// TIA Portal V20 export
TYPE "UDT_Service_ValueDefinition"
   STRUCT
      indexMTP : Int;   // Index of value / MTP Index of value
      indexIO : Int;   // Index of value / IO Index of value
      "type" : Int;   // Type of parameter
      controlModule : Byte := 16#FF;   // Number of control module used with parameter
   END_STRUCT;
END_TYPE
